Yaskawa INFORM job: Flat1.JBI

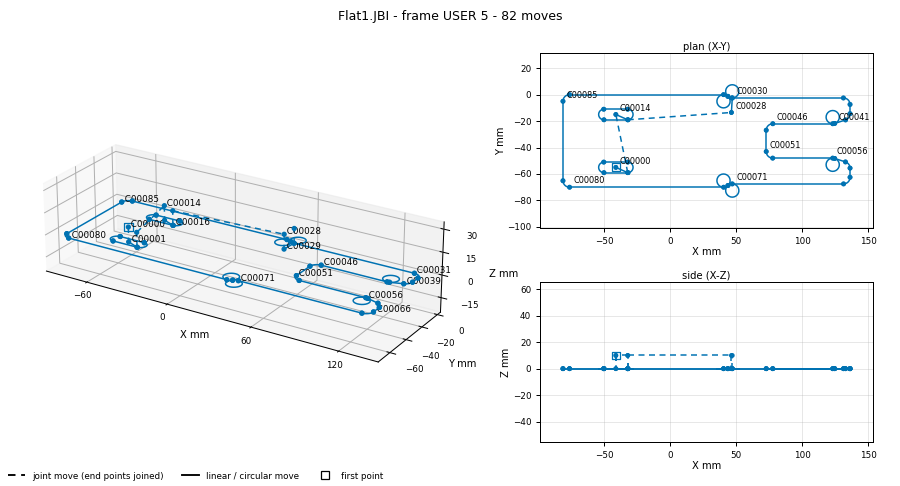
[picture p0: tool path of Flat1.JBI in frame USER 5, 82 of 102 moves have a stored position in this frame; points joined in program order, loops and branches not executed]
/JOB
//NAME FLAT1
//POS
///NPOS 102,0,0,0,0,0
///TOOL 1
///USER 5
///POSTYPE USER
///RECTAN
///RCONF 1,0,0,0,0,0,0,0,0,0,0,0,0,0,0,0,0,0,0,0,0,0,0,0
C00000=-41.059,-55.0,10.0,0,0,0
C00001=-41.059,-55.0,0.0,0,0,0
C00002=-32.059,-59.0,0.0,0,0,0
C00003=-50.059,-59.0,0.0,0,0,0
C00004=-50.059,-59.0,0.0,0,0,0
C00005=-50.216,-58.997,0.0,0,0,0
C00006=-50.373,-51.012,0.0,0,0,0
C00007=-50.059,-51.0,0.0,0,0,0
C00008=-32.059,-51.0,0.0,0,0,0
C00009=-32.059,-51.0,0.0,0,0,0
C00010=-31.902,-51.003,0.0,0,0,0
C00011=-31.745,-58.988,0.0,0,0,0
C00012=-32.059,-59.0,0.0,0,0,0
C00013=-32.059,-59.0,10.0,0,0,0
C00014=-41.059,-15.0,10.0,0,0,0
C00015=-41.059,-15.0,0.0,0,0,0
C00016=-32.059,-19.0,0.0,0,0,0
C00017=-50.059,-19.0,0.0,0,0,0
C00018=-50.059,-19.0,0.0,0,0,0
C00019=-50.216,-18.997,0.0,0,0,0
C00020=-50.373,-11.012,0.0,0,0,0
C00021=-50.059,-11.0,0.0,0,0,0
C00022=-32.059,-11.0,0.0,0,0,0
C00023=-32.059,-11.0,0.0,0,0,0
C00024=-31.902,-11.003,0.0,0,0,0
C00025=-31.745,-18.988,0.0,0,0,0
C00026=-32.059,-19.0,0.0,0,0,0
C00027=-32.059,-19.0,10.0,0,0,0
C00028=46.337,-13.481,10.0,0,0,0
C00029=46.337,-13.481,0.0,0,0,0
C00030=46.99,-2.5,0.0,0,0,0
C00031=131.059,-2.5,0.0,0,0,0
C00032=131.059,-2.5,0.0,0,0,0
C00033=134.663,-4.034,0.0,0,0,0
C00034=136.055,-7.304,0.0,0,0,0
C00035=136.059,-7.5,0.0,0,0,0
C00036=136.059,-14.367,0.0,0,0,0
C00037=136.059,-14.367,0.0,0,0,0
C00038=133.934,-18.458,0.0,0,0,0
C00039=132.753,-19.072,0.0,0,0,0
C00040=132.604,-19.123,0.0,0,0,0
C00041=124.501,-21.755,0.0,0,0,0
C00042=124.501,-21.755,0.0,0,0,0
C00043=127.891,-17.802,0.0,0,0,0
C00044=122.996,-22.0,0.0,0,0,0
C00045=122.956,-22.0,0.0,0,0,0
C00046=77.66,-22.0,0.0,0,0,0
C00047=77.66,-22.0,0.0,0,0,0
C00048=74.056,-23.534,0.0,0,0,0
C00049=72.664,-26.804,0.0,0,0,0
C00050=72.66,-27.0,0.0,0,0,0
C00051=72.66,-43.0,0.0,0,0,0
C00052=72.66,-43.0,0.0,0,0,0
C00053=74.194,-46.604,0.0,0,0,0
C00054=77.464,-47.996,0.0,0,0,0
C00055=77.66,-48.0,0.0,0,0,0
C00056=122.956,-48.0,0.0,0,0,0
C00057=122.956,-48.0,0.0,0,0,0
C00058=127.897,-52.237,0.0,0,0,0
C00059=124.464,-48.233,0.0,0,0,0
C00060=124.501,-48.245,0.0,0,0,0
C00061=132.604,-50.877,0.0,0,0,0
C00062=132.604,-50.877,0.0,0,0,0
C00063=134.06,-51.633,0.0,0,0,0
C00064=136.057,-55.476,0.0,0,0,0
C00065=136.059,-55.633,0.0,0,0,0
C00066=136.059,-62.5,0.0,0,0,0
C00067=136.059,-62.5,0.0,0,0,0
C00068=134.525,-66.104,0.0,0,0,0
C00069=131.255,-67.496,0.0,0,0,0
C00070=131.059,-67.5,0.0,0,0,0
C00071=46.99,-67.5,0.0,0,0,0
C00072=46.99,-67.5,0.0,0,0,0
C00073=42.297,-70.774,0.0,0,0,0
C00074=43.751,-68.691,0.0,0,0,0
C00075=43.683,-68.75,0.0,0,0,0
C00076=43.683,-68.75,0.0,0,0,0
C00077=45.037,-66.81,0.0,0,0,0
C00078=40.466,-69.999,0.0,0,0,0
C00079=40.376,-70.0,0.0,0,0,0
C00080=-76.059,-70.0,0.0,0,0,0
C00081=-76.059,-70.0,0.0,0,0,0
C00082=-79.663,-68.466,0.0,0,0,0
C00083=-81.055,-65.196,0.0,0,0,0
C00084=-81.059,-65.0,0.0,0,0,0
C00085=-81.059,-5.0,0.0,0,0,0
C00086=-81.059,-5.0,0.0,0,0,0
C00087=-79.525,-1.396,0.0,0,0,0
C00088=-76.255,-0.004,0.0,0,0,0
C00089=-76.059,0.0,0.0,0,0,0
C00090=40.376,0.0,0.0,0,0,0
C00091=40.376,0.0,0.0,0,0,0
C00092=45.069,-3.274,0.0,0,0,0
C00093=43.615,-1.191,0.0,0,0,0
C00094=43.683,-1.25,0.0,0,0,0
C00095=43.683,-1.25,0.0,0,0,0
C00096=42.329,0.69,0.0,0,0,0
C00097=46.9,-2.499,0.0,0,0,0
C00098=46.99,-2.5,0.0,0,0,0
C00099=46.99,-2.5,10.0,0,0,0
///POSTYPE PULSE
///PULSE
C00100=0,0,0,0,0,0
C00101=0,0,0,0,0,0
//INST
///DATE 2025/08/07 16:41
///ATTR SC,RW,RJ
////FRAME USER 5
///GROUP1 RB1
NOP
DOUT OT#(1) OFF
MOVJ C00101 VJ=10.0
DOUT OT#(1) OFF
TIMER T=0.50
MOVJ C00000 VJ=10.0
MOVJ C00001 VJ=10.0
DOUT OT#(1) ON
TIMER T=0.50
MOVL C00002 V=38.0
MOVL C00003 V=38.0
MOVC C00004 V=38.0
MOVC C00005 V=38.0
MOVC C00006 V=38.0 FPT
MOVL C00007 V=38.0
MOVL C00008 V=38.0
MOVC C00009 V=38.0
MOVC C00010 V=38.0
MOVC C00011 V=38.0 FPT
MOVL C00012 V=38.0
DOUT OT#(1) OFF
TIMER T=0.50
MOVJ C00013 VJ=10.0
MOVJ C00014 VJ=10.0
MOVJ C00015 VJ=10.0
DOUT OT#(1) ON
TIMER T=0.50
MOVL C00016 V=38.0
MOVL C00017 V=38.0
MOVC C00018 V=38.0
MOVC C00019 V=38.0
MOVC C00020 V=38.0 FPT
MOVL C00021 V=38.0
MOVL C00022 V=38.0
MOVC C00023 V=38.0
MOVC C00024 V=38.0
MOVC C00025 V=38.0 FPT
MOVL C00026 V=38.0
DOUT OT#(1) OFF
TIMER T=0.50
MOVJ C00027 VJ=10.0
MOVJ C00028 VJ=10.0
MOVJ C00029 VJ=10.0
DOUT OT#(1) ON
TIMER T=0.50
MOVL C00030 V=38.0
MOVL C00031 V=38.0
MOVC C00032 V=38.0
MOVC C00033 V=38.0
MOVC C00034 V=38.0 FPT
MOVL C00035 V=38.0
MOVL C00036 V=38.0
MOVC C00037 V=38.0
MOVC C00038 V=38.0
MOVC C00039 V=38.0 FPT
MOVL C00040 V=38.0
MOVL C00041 V=38.0
MOVC C00042 V=38.0
MOVC C00043 V=38.0
MOVC C00044 V=38.0 FPT
MOVL C00045 V=38.0
MOVL C00046 V=38.0
MOVC C00047 V=38.0
MOVC C00048 V=38.0
MOVC C00049 V=38.0 FPT
MOVL C00050 V=38.0
MOVL C00051 V=38.0
MOVC C00052 V=38.0
MOVC C00053 V=38.0
MOVC C00054 V=38.0 FPT
MOVL C00055 V=38.0
MOVL C00056 V=38.0
MOVC C00057 V=38.0
MOVC C00058 V=38.0
MOVC C00059 V=38.0 FPT
MOVL C00060 V=38.0
MOVL C00061 V=38.0
MOVC C00062 V=38.0
MOVC C00063 V=38.0
MOVC C00064 V=38.0 FPT
MOVL C00065 V=38.0
MOVL C00066 V=38.0
MOVC C00067 V=38.0
MOVC C00068 V=38.0
MOVC C00069 V=38.0 FPT
MOVL C00070 V=38.0
MOVL C00071 V=38.0
MOVC C00072 V=38.0
MOVC C00073 V=38.0
MOVC C00074 V=38.0 FPT
MOVL C00075 V=38.0
MOVC C00076 V=38.0
MOVC C00077 V=38.0
MOVC C00078 V=38.0 FPT
MOVL C00079 V=38.0
MOVL C00080 V=38.0
MOVC C00081 V=38.0
MOVC C00082 V=38.0
MOVC C00083 V=38.0 FPT
MOVL C00084 V=38.0
MOVL C00085 V=38.0
MOVC C00086 V=38.0
MOVC C00087 V=38.0
MOVC C00088 V=38.0 FPT
MOVL C00089 V=38.0
MOVL C00090 V=38.0
MOVC C00091 V=38.0
MOVC C00092 V=38.0
MOVC C00093 V=38.0 FPT
MOVL C00094 V=38.0
MOVC C00095 V=38.0
MOVC C00096 V=38.0
MOVC C00097 V=38.0 FPT
MOVL C00098 V=38.0
DOUT OT#(1) OFF
TIMER T=0.50
MOVJ C00099 VJ=10.0
DOUT OT#(1) OFF
MOVJ C00100 VJ=10.0
END
